(* IEC 61131-3 sources: ICSQuartz/benchmarks/oscat_basic_charname/src, 1 file *)

(* ---- program.st ---- *)
PROGRAM PLC_PRG
VAR_INPUT
    in_c: BYTE;
END_VAR

CHARNAME(in_c);

END_PROGRAM
